pPts^.ctrl.fbPts_Mdc_Umc.iniAllCtrlArrays(pCtrlInst,pCtrlCIf,pPts^.id.Pts_Mdc_Umc);
pPts^.ctrl.fbPts_Mdc.iniAllCtrlArrays(pCtrlInst,pCtrlCIf,pPts^.id.Pts_Mdc);
pPts^.ctrl.fbPts_Mdc.Drive := ADR(pPts^.ctrl.fbPts_Mdc_Umc);

pPts^.ctrl.fbPts_RAX.iniAllCtrlArrays(pCtrlInst,pCtrlCIf,pPts^.id.Pts_RAX);
pPts^.ctrl.fbPts_RAX.In_pAD_SIf:= pPts^.ctrl.fbPts_RAX_POD.AD_SIf;	

pPts^.ctrl.fbPts.iniAllCtrlArrays(pCtrlInst,pCtrlCIf,pPts^.id.Pts);
pPts^.ctrl.fbPts.Belt := ADR(pPts^.ctrl.fbPts_Ptb);
pPts^.ctrl.fbPts.Malteser := ADR(pPts^.ctrl.fbPts_Mdc);
pPts^.ctrl.fbPts.Servo := ADR(pPts^.ctrl.fbPts_RAX);
                
END_FUNCTION

FUNCTION_BLOCK FB_OvenSendDch EXTENDS FB_DataChannelSendBase IMPLEMENTS I_DataChannelSend
  VAR
    m_pOutputData : POINTER TO T_Oven_DCH;  (* Saber Inteface Variables ----------------------------------------------------------------- *)
  END_VAR

                  SUPER^();
                

{attribute 'object_name' := 'SendData'}
METHOD SendData : BOOL
  VAR_INPUT
    udiDataSize : UDINT;
    pData : POINTER TO BYTE;
  END_VAR
                        SendData := FALSE;

IF m_eState = E_PlcSaberDHCState.WaitForJob THEN
	IF (udiDataSize > 0 ) AND (pData <> TC3_MEMMAN.NULL) THEN
		TC2_SYSTEM.MEMCPY(destAddr := m_pOutputData, srcAddr := pData, n := udiDataSize);
		m_eState := E_PlcSaberDHCState.SendData;	
		SendData := TRUE;
	END_IF	
END_IF
                      
END_METHOD

{attribute 'object_name' := 'InitChannel'}
METHOD InitChannel : BOOL
  VAR_INPUT
    udiDataSize : UDINT;
    pOutputData : POINTER TO BYTE;
  END_VAR
                        InitChannel := FALSE;

IF udiDataSize > 0 THEN
	IF pOutputData <> TC3_MEMMAN.NULL THEN
		m_uinDataSize := udiDataSize;
		m_pOutputData := pOutputData;
		m_eState := E_PlcSaberDHCState.Init;
		InitChannel := TRUE;
	END_IF
END_IF

                      
END_METHOD
END_FUNCTION_BLOCK

CONFIGURATION Application
  RESOURCE BasePpt ON PLC
    VAR_GLOBAL CONSTANT  (* Constants *)
      MAX_INT : INT := 32767;  (* Oven ---------------------------------------------------------------------- *)
      MIN_INT : INT := -32768;
      MAX_NUMBER_OF_OVEN_MODULES : UINT := 8;
      WRITE_BUFFER_LENGTH : UDINT := 98;
      READ_BUFFER_LENGTH : UDINT := 103;
    END_VAR
    VAR_GLOBAL CONSTANT  (* Global_Version - This function has been automatically generated from the project information. *)
      {attribute 'const_non_replaced'}
      stLibVersion_BasePpt : ST_LibVersion := (iMajor := 0, iMinor := 0, iBuild := 0, iRevision := 89, sVersion := '0.0.0.89');
    END_VAR
    VAR_GLOBAL CONSTANT  (* IBH_CmdState *)
      cCMD_CONNECT : INT := 202;  (* ctrl commands definitions specific commands >200 - every command has to be a even number *)
      cCMD_WRITE : INT := 204;
      cCMD_READ : INT := 206;
      cCMD_DISCONNECT : INT := 208;
      cSTA_CONNECTBusy : INT := 201;  (* ctrl specific states definitions *)
      cSTA_CONNECT : INT := 202;
      cSTA_WRITEBusy : INT := 203;
      cSTA_WRITE : INT := 204;
      cSTA_READBusy : INT := 205;
      cSTA_READ : INT := 206;
      cSTA_DISCONNECTBusy : INT := 207;
      cSTA_DISCONNECT : INT := 208;
      cSTA_SUB_1 : INT := 301;
      cSTA_SUB_2 : INT := 302;
      cSTA_SUB_3 : INT := 303;
      cSTA_SUB_4 : INT := 304;
      cSTA_SUB_5 : INT := 305;
    END_VAR
    VAR_GLOBAL CONSTANT  (* POD_Cmd *)
      cPOD_STA_PowerOff : INT := 0;  (* Switch controller on *)
      cPOD_STA_Error : INT := 256;  (* Error *)
      cPOD_STA_WaitForJob : INT := 1000;
      cPOD_STA_PowerOnBusy : INT := 1001;
      cPOD_STA_HomeBusy : INT := 1006;  (* Homing *)
      cPOD_STA_RelMoveBusy : INT := 1007;  (* Start move with relative move distance *)
      cPOD_STA_AbsMoveBusy : INT := 1010;  (* Start move with absolute target position *)
      cPOD_STA_PosMoveBusy : INT := 1011;  (* Start move in positive direction *)
      cPOD_STA_PosMove : INT := 1012;
      cPOD_STA_NegMoveBusy : INT := 1013;  (* Start move in negative direction *)
      cPOD_STA_NegMove : INT := 1014;
      cPOD_STA_StopBusy : INT := 1015;  (* controller on standstill *)
      cPOD_STA_QStopBusy : INT := 1017;  (* controller on standstill *)
      cPOD_STA_NegJogBusy : INT := 1019;  (* controller on standstill *)
      cPOD_STA_PosJogBusy : INT := 1021;  (* controller on standstil *)
      cPOD_STA_ModMoveBusy : INT := 1023;
      cPOD_STA_ModMove : INT := 1024;
      cPOD_STA_StorePara : INT := 1050;
      cPOD_STA_WritePara : INT := 1052;
      cPOD_CMD_DONE : INT := -1;  (* ctrl commands definitions specific commands >200 - every command has to be a even number *)
      cPOD_CMD_CTRL_ON : INT := 1002;  (* Switch controller on *)
      cPOD_CMD_CTRL_OFF : INT := 1004;  (* Switch controller off *)
      cPOD_CMD_HOME : INT := 1006;  (* Homing *)
      cPOD_CMD_REL_MOVE : INT := 1008;  (* Start move with relative move distance *)
      cPOD_CMD_ABS_MOVE : INT := 1010;  (* Start move with absolute target position *)
      cPOD_CMD_POS_MOVE : INT := 1012;  (* Start move in positive direction *)
      cPOD_CMD_NEG_MOVE : INT := 1014;  (* Start move in negative direction *)
      cPOD_CMD_STOP : INT := 1016;  (* Stop movement with controller on *)
      cPOD_CMD_EMCY_STOP_CTRL_OFF : INT := 1018;  (* Emergency stop with controller off *)
      cPOD_CMD_POS_JOG : INT := 1020;  (* Start move in positive direction *)
      cPOD_CMD_NEG_JOG : INT := 1022;
      cPOD_CMD_MOD_MOVE : INT := 1024;  (* Start move with modulo positionining (based on modulofactor defined in axis parameter!) *)
      cPOD_CMD_STORE_PARAMETER : INT := 1050;
      cPOD_CMD_WRITE_PARAMETER : INT := 1052;
      cPOD_SCMD_WRITE_PARA : INT := 2002;  (* Service Jobs (parallel to active job) *)
      cPOD_SCMD_READ_PARA : INT := 2004;
      cPOD_SCMD_RESET_ABSENCODER : INT := 2006;
      cPOD_SCMD_WRITE_PARA_NC : INT := 2008;
      cPOD_SCMD_READ_PARA_NC : INT := 2010;
    END_VAR
    VAR_GLOBAL CONSTANT  (* TCP_CmdState *)
      cCMD_Close : INT := 202;  (* ctrl commands definitions specific commands >200 - every command has to be a even number *)
      cCMD_Connect : INT := 204;
      cSTA_CloseBusy : INT := 201;  (* ctrl specific states definitions *)
      cSTA_Close : INT := 202;
      cSTA_ConnectBusy : INT := 203;
      cSTA_Connect : INT := 204;
    END_VAR
    VAR_GLOBAL CONSTANT  (* TCP_Constants *)
      MAX_DATASET_SIZE : UDINT := 900;  (* Define length of data buffer. Max. 900 Byte *)
    END_VAR
    VAR_GLOBAL CONSTANT  (* JCL_CmdState *)
      cCMD_Standby : INT := 202;  (* Preparing jetter for production *)
      cCMD_Calibration : INT := 204;  (* Start calibration routine for MM camera system *)
      cCMD_CleanPrintHeads : INT := 206;  (* Start automatic cleaning cycle for both printheads *)
      cCMD_ResetAlarm : INT := 230;  (* Reset pending alarms *)
      cCMD_RequestState : INT := 240;  (* Send back the state msg. *)
      cSTA_StandbyBusy : INT := 201;  (* ctrl specific states definitions *)
      cSTA_Standby : INT := cCMD_Standby;
      cSTA_ConnectBusy : INT := 250;
      cSTA_CleanPrintHeadsBusy : INT := 205;
      cSTA_CleanPrintHeads : INT := cCMD_CleanPrintHeads;
      cSTA_CalibrationBusy : INT := 203;
      cSTA_Calibration : INT := cCMD_Calibration;
      cSTA_ParkBusy : INT := 211;
      cSTA_MaintenanceBusy : INT := 208;
      cSTA_MaintenanceInWork : INT := 209;
      cSTA_MaintenanceDone : INT := 210;
      cSTA_MANUALMODE : INT := 212;
      cSUB_WaitingForConnection : INT := 300;  (* sub states *)
      cSUB_WaitingForState : INT := 301;
      cSUB_WaitingSocketClosed : INT := 302;
      cSUB_SendPon : INT := 303;
      cSUB_Done : INT := 999;
      cSUB_WaitForCleaningToStart : INT := 304;
      cSUB_CleaningBusy : INT := 305;
    END_VAR
    VAR_GLOBAL CONSTANT  (* JCL_Constants *)
      JCL_MsgId_Command : UINT := 1;  (* MsgID (valid for jetter TCP server protocol) *)
      JCL_MsgId_State : UINT := 2;
      JCL_MsgId_Alarm : UINT := 4;
      JCL_MsgId_PrintDone : UINT := 5;
      JCL_MsgId_ReqCleaning : UINT := 6;
      JCL_CMD_PowerOn : USINT := 2;  (* Jetter CMD (valid for jetter TCP server protocol) *)
      JCL_CMD_Off : USINT := 6;
      JCL_STA_Standby : USINT := 202;
      JCL_CMD_Standby : USINT := 202;
      JCL_CMD_Run : USINT := 10;
      JCL_CMD_CleanPrintHeads : USINT := 206;
      JCL_CMD_Calibration : USINT := 204;
      JCL_CMD_ResetAlarm : USINT := 230;
      JCL_CMD_RequestState : USINT := 240;
    END_VAR
    VAR_GLOBAL CONSTANT  (* RAX_CmdState *)
      cCMD_HOME : INT := 202;  (* ctrl commands definitions specific commands >200 - every command has to be a even number *)
      cCMD_POS : INT := 204;
      cCMD_JOG_NEG : INT := 210;
      cCMD_JOG_POS : INT := 212;
      cCMD_REL_POS : INT := 214;
      cCMD_TURN : INT := 216;
      cSTA_POSBusy : INT := 203;  (* ctrl specific states definitions *)
      cSTA_POS : INT := RAX_CmdState.cCMD_POS;
      cSTA_REL_POSBusy : INT := 213;
      cSTA_REL_POS : INT := RAX_CmdState.cCMD_REL_POS;
      cSTA_JOG_NEG : INT := RAX_CmdState.cCMD_JOG_NEG;
      cSTA_JOG_POS : INT := RAX_CmdState.cCMD_JOG_POS;
      cSTA_TURNBusy : INT := 215;
      cSTA_TURN : INT := RAX_CmdState.cCMD_TURN;
    END_VAR
    VAR_GLOBAL CONSTANT  (* BCH_CmdState *)
      cCMD_READ : INT := 200;
      cCMD_TESTSEQUENCE : INT := 202;
      cSTA_TESTSEQUENCE : INT := 202;
      cSUB_WAITPAPER : INT := 300;
      cSUB_BARCODEREADstart : INT := 310;
      cSUB_BARCODREREADbusy : INT := 311;
      cSUB_BARCODREREAD : INT := 312;
      cSUB_WAITPAPERGONE : INT := 313;
      cSUB_WAITPAPERGONEDELAY : INT := 314;
    END_VAR
    VAR_GLOBAL CONSTANT  (* MDC_CmdState *)
      cCMD_INITIALIZE : INT := 202;  (* ctrl commands definitions specific commands >200 - every command has to be a even number *)
      cCMD_TURN : INT := 204;
      cCMD_PREPOSITION : INT := 210;
      cSTA_InitializeBusy : INT := 201;  (* ctrl specific states definitions *)
      cSTA_InPositionBusy : INT := 203;
      cSTA_InPosition : INT := 205;
      cSTA_StartTurnBusy : INT := 207;
      cSTA_TurnBusy : INT := 209;
      cSTA_PREPOSITIONbusy : INT := 220;
      cSTA_PREPOSITION : INT := 221;
      cSTA_TURNDONE : INT := 222;
      cSUB_TURNbusy : INT := 300;
      cSUB_STOPbusy : INT := 301;
      cSUB_FINDHOLEbusy : INT := 302;
    END_VAR
    VAR_GLOBAL CONSTANT  (* OVN_CmdState *)
      cCMD_BELTONLY : INT := 202;  (* ctrl commands definitions specific commands >200 - every command has to be a even number *)
      cSTA_BELTONLYBusy : INT := 201;  (* ctrl specific states definitions *)
      cSTA_BELTONLY : INT := 202;
      cSUB_WAITOFF : INT := 300;
      cSUB_WAITPAPER : INT := 301;
      cSUB_DONE : INT := 302;
    END_VAR
    VAR_GLOBAL CONSTANT  (* PTB_CmdState *)
      cCMD_EJECTPAPER : INT := 202;  (* ctrl commands definitions *)
      cCMD_STACKPAPER : INT := 204;
      cSTA_EJECTPAPERbusy : INT := 201;  (* specific commands >200 - every command has to be a even number ctrl specific states definitions *)
      cSTA_EJECTPAPER : INT := 202;
      cSTA_STACKPAPERbusy : INT := 203;
      cSTA_STACKPAPER : INT := 204;
      cSUB_EMPTYstart : INT := 300;  (* ctrl specific sub states definitions *)
      cSUB_EMPTYWAITPAPERbusy : INT := 301;
      cSUB_EMPTYWAITPAPERdebounce : INT := 302;
      cSUB_EMPTYWAITPAPERGONEbusy : INT := 303;
      cSUB_EMPTYWAITPAPERGONEdebounce : INT := 304;
      cSUB_EMPTYWAITDRIVESTOPED : INT := 305;
      cSUB_WAITPAPER : INT := 306;
      cSUB_WAITPAPERGONE : INT := 307;
      cSUB_STARTSTACKDELAY : INT := 308;
      cSUB_PAPERDISTANCEstart : INT := 309;
      cSUB_PAPERDISTANCEbusy : INT := 310;
      cSUB_PAPERDISTANCESTOPbusy : INT := 311;
      cSUB_STARTENTRYDRIVEbusy : INT := 312;
      cSUB_STARTENTRYDRIVE : INT := 313;
    END_VAR
    VAR_GLOBAL CONSTANT  (* PBC_CmdState *)
      cCMD_SINGLE : INT := 202;  (* ctrl specific command definitions *)
      cCMD_MANUALSTART : INT := 204;
      cSTA_INITbusy : INT := 205;  (* ctrl specific states definitions *)
      cSUB_WAITPAPER : INT := 300;
      cSUB_POSITIONbusy : INT := 301;
      cSUB_POSITIONSTOPbusy : INT := 302;
      cSUB_EVALUATEEJECT : INT := 303;
      cSUB_EJECTbusy : INT := 304;
      cSUB_EJECTSTOPbusy : INT := 305;
      cSUB_POSITIONSTARTbusy : INT := 306;
      cSUB_EJECTSTARTbusy : INT := 307;
      cSUB_READYEJECT : INT := 308;
      cSUB_WAITPAPERGONETABLE : INT := 309;
      cSUB_POSITIONRETRYDELAY : INT := 313;  (* cSUB_BARCODEREADstart : INT := 310; cSUB_BARCODREREADbusy : INT := 311; cSUB_BARCODREREAD : INT := 312; *)
      cSUB_POSITIONRETRYSTOP : INT := 314;
    END_VAR
    VAR_GLOBAL CONSTANT  (* PCE_CmdState *)
      cSUB_PAPERENTRY : INT := 300;  (* ctrl commands definitions specific commands >200 - every command has to be a even number ctrl specific states definitions *)
      cSUB_PAPERENTRYDelay : INT := 301;
      cSUB_PAPEREXIT : INT := 302;
    END_VAR
    VAR_GLOBAL CONSTANT  (* PST_CmdState *)
      cCMD_EJECT : INT := 202;  (* specific commands >200 - every command has to be a even number ctrl commands definitions *)
      cSTA_EJECTbusy : INT := 201;  (* main states *)
      cSUB_WAITNEWPAPERDETECTED : INT := 300;  (* sub states *)
      cSUB_DELAYREADBARCODEBusy : INT := 301;
      cSUB_RETRYREADBARCODE : INT := 302;
      cSUB_READBARCODEbusy : INT := 303;
      cSUB_CHECKEJECTCONDITIONS : INT := 304;
      cSUB_DELAYSTACKEJECTBusy : INT := 305;
      cSUB_MOVEBELTEJECTDIRECTIONBusy : INT := 306;
      cSUB_STOPBELTBusy : INT := 307;
      cSUB_WAITBEFOREMOVINGREVERSE : INT := 308;
      cSUB_MOVEBELTREVERSEBusy : INT := 309;
      cSUB_DONE : INT := 999;
    END_VAR
    VAR_GLOBAL CONSTANT  (* PTS_CmdState *)
      cCMD_TURN : INT := 202;  (* ctrl specific command definitions *)
      cCMD_STANDBY : INT := 204;
      cSTA_STANDBYBusy : INT := 203;  (* ctrl specific states definitions *)
      cSTA_STANDBY : INT := 204;
      cSTA_PaperDelayBusy : INT := 205;
      cSTA_TurnPaperBusy : INT := 207;
      cSTA_WaitPaperGone : INT := 209;
      cSTA_EmptyDelayBusy : INT := 211;
      cSTA_TurnEmptyBusy : INT := 213;
      cSTA_InitializeBusy : INT := 215;
      cSTA_WaitPaper : INT := 217;
      cSTA_GetItemBusy : INT := 219;
      cSUB_WAIT_START : INT := 300;  (* ctrl specific substates definitions *)
      cSUB_WAIT_DONE : INT := 301;
      cSUB_TURNbusy : INT := 302;
      cSUB_TURNDONE : INT := 303;
      cSUB_PREPOSITIONbusy : INT := 304;
      cSUB_DELAYbusy : INT := 305;
      cSUB_WAITPAPERGONEbusy : INT := 306;
      cPTS_MAX_AUTOPOS : UINT := 5;  (* Other Constants *)
      cPTS_MAX_DISTRIBUTION : INT := 2;
    END_VAR
    VAR_GLOBAL  (* PTS_Persistent *)
      udiPTS_Counter_Persistent : UDINT;  (* Count of turn movements. This is a persistent variable, reset only with reset origin *)
    END_VAR
    VAR_GLOBAL CONSTANT  (* LUT_Constants *)
      MaxLookupSize : INT := 20;  (* max size of lookup table *)
    END_VAR
    VAR_GLOBAL CONSTANT  (* OvenConst *)
      cRECVDATACHANNELBUFFER : INT := 20;
    END_VAR
  END_RESOURCE
END_CONFIGURATION
